FUNCTION_BLOCK FB_System_WDT_500

VAR_INPUT
	Betrieb_Anford_auto				: BOOL;
	Freigabe_Deakt_auto 			: BOOL;
	Regelung_Modus_auto				: USINT;
	Regelung_Nachtabs_auto			: BOOL;
	Regelung_Sollw_auto				: REAL;
	Temp_Rueckl_Wand_Ost_Sektor1	: REAL;
	Temp_Rueckl_Wand_Ost_Sektor2	: REAL;
	Temp_Rueckl_Wand_Ost_Sektor3	: REAL;
	Temp_Rueckl_Wand_West_Sektor1	: REAL;
	Temp_Rueckl_Wand_West_Sektor2	: REAL;
	Temp_Rueckl_Wand_West_Sektor3	: REAL;
	Temp_Rueckl_Decke_Ost_Sektor1	: REAL;
	Temp_Rueckl_Decke_Ost_Sektor2	: REAL;
	Temp_Rueckl_Decke_Ost_Sektor3	: REAL;
	Temp_Rueckl_Decke_West_Sektor1	: REAL;
	Temp_Rueckl_Decke_West_Sektor2	: REAL;
	Temp_Rueckl_Decke_West_Sektor3	: REAL;
	Temp_Rueckl_Aussen_Ost			: REAL;
	Temp_Rueckl_Aussen_West			: REAL;
	Temp_AFA_Aussen					: REAL;

END_VAR
VAR_OUTPUT
	{attribute 'OPC.UA.DA' := '1'}Steuerung				: ST_System_WDT_Steuerung;		
	{attribute 'OPC.UA.DA' := '1'}Stellwert				: ST_System_WDT_Stellwert;		
	{attribute 'OPC.UA.DA' := '1'}Zustand					: ST_System_WDT_Zustand;	
	{attribute 'OPC.UA.DA' := '1'}Parameter				: ST_System_WDT_Parameter;		
END_VAR
VAR
	Pumpe_405				: FB_PU;
	Stellventil_401_402		: FB_SVs;
	Stellventil_403_404		: FB_SVs;
	Stellventil_504_505		: FB_SVs_504_505;
	Pumpe_500				: FB_PU;
	Regelventil_500			: FB_RV;
	Regelventil_561			: FB_RV;
	Regelventil_562			: FB_RV;
	Regelventil_563			: FB_RV;
	Regelventil_571			: FB_RV;
	Regelventil_572			: FB_RV;
	Regelventil_573			: FB_RV;
	Regelventil_541			: FB_RV;
	Regelventil_542			: FB_RV;
	Regelventil_543			: FB_RV;
	Regelventil_551			: FB_RV;
	Regelventil_552			: FB_RV;
	Regelventil_553			: FB_RV;

	Zustandscheck			: FB_System_WDT_Zustandscheck;
	Logik					: FB_System_WDT_Logik;
	Ablaufsteuerung			: FB_System_WDT_Ablaufsteuerung;
	Sollwertscheck			: FB_System_WDT_Sollwertscheck;
	Regelung				: FB_System_WDT_Regelung;
	Stellwertscheck			: FB_System_WDT_Stellwertscheck;




END_VAR
VAR // added by the converter: edge detectors and wires of the graphical bodies
    _w1, _w2, _w4, _w6, _w7, _w8, _w9 : ANY;
    _w3, _w5 : BOOL;
END_VAR

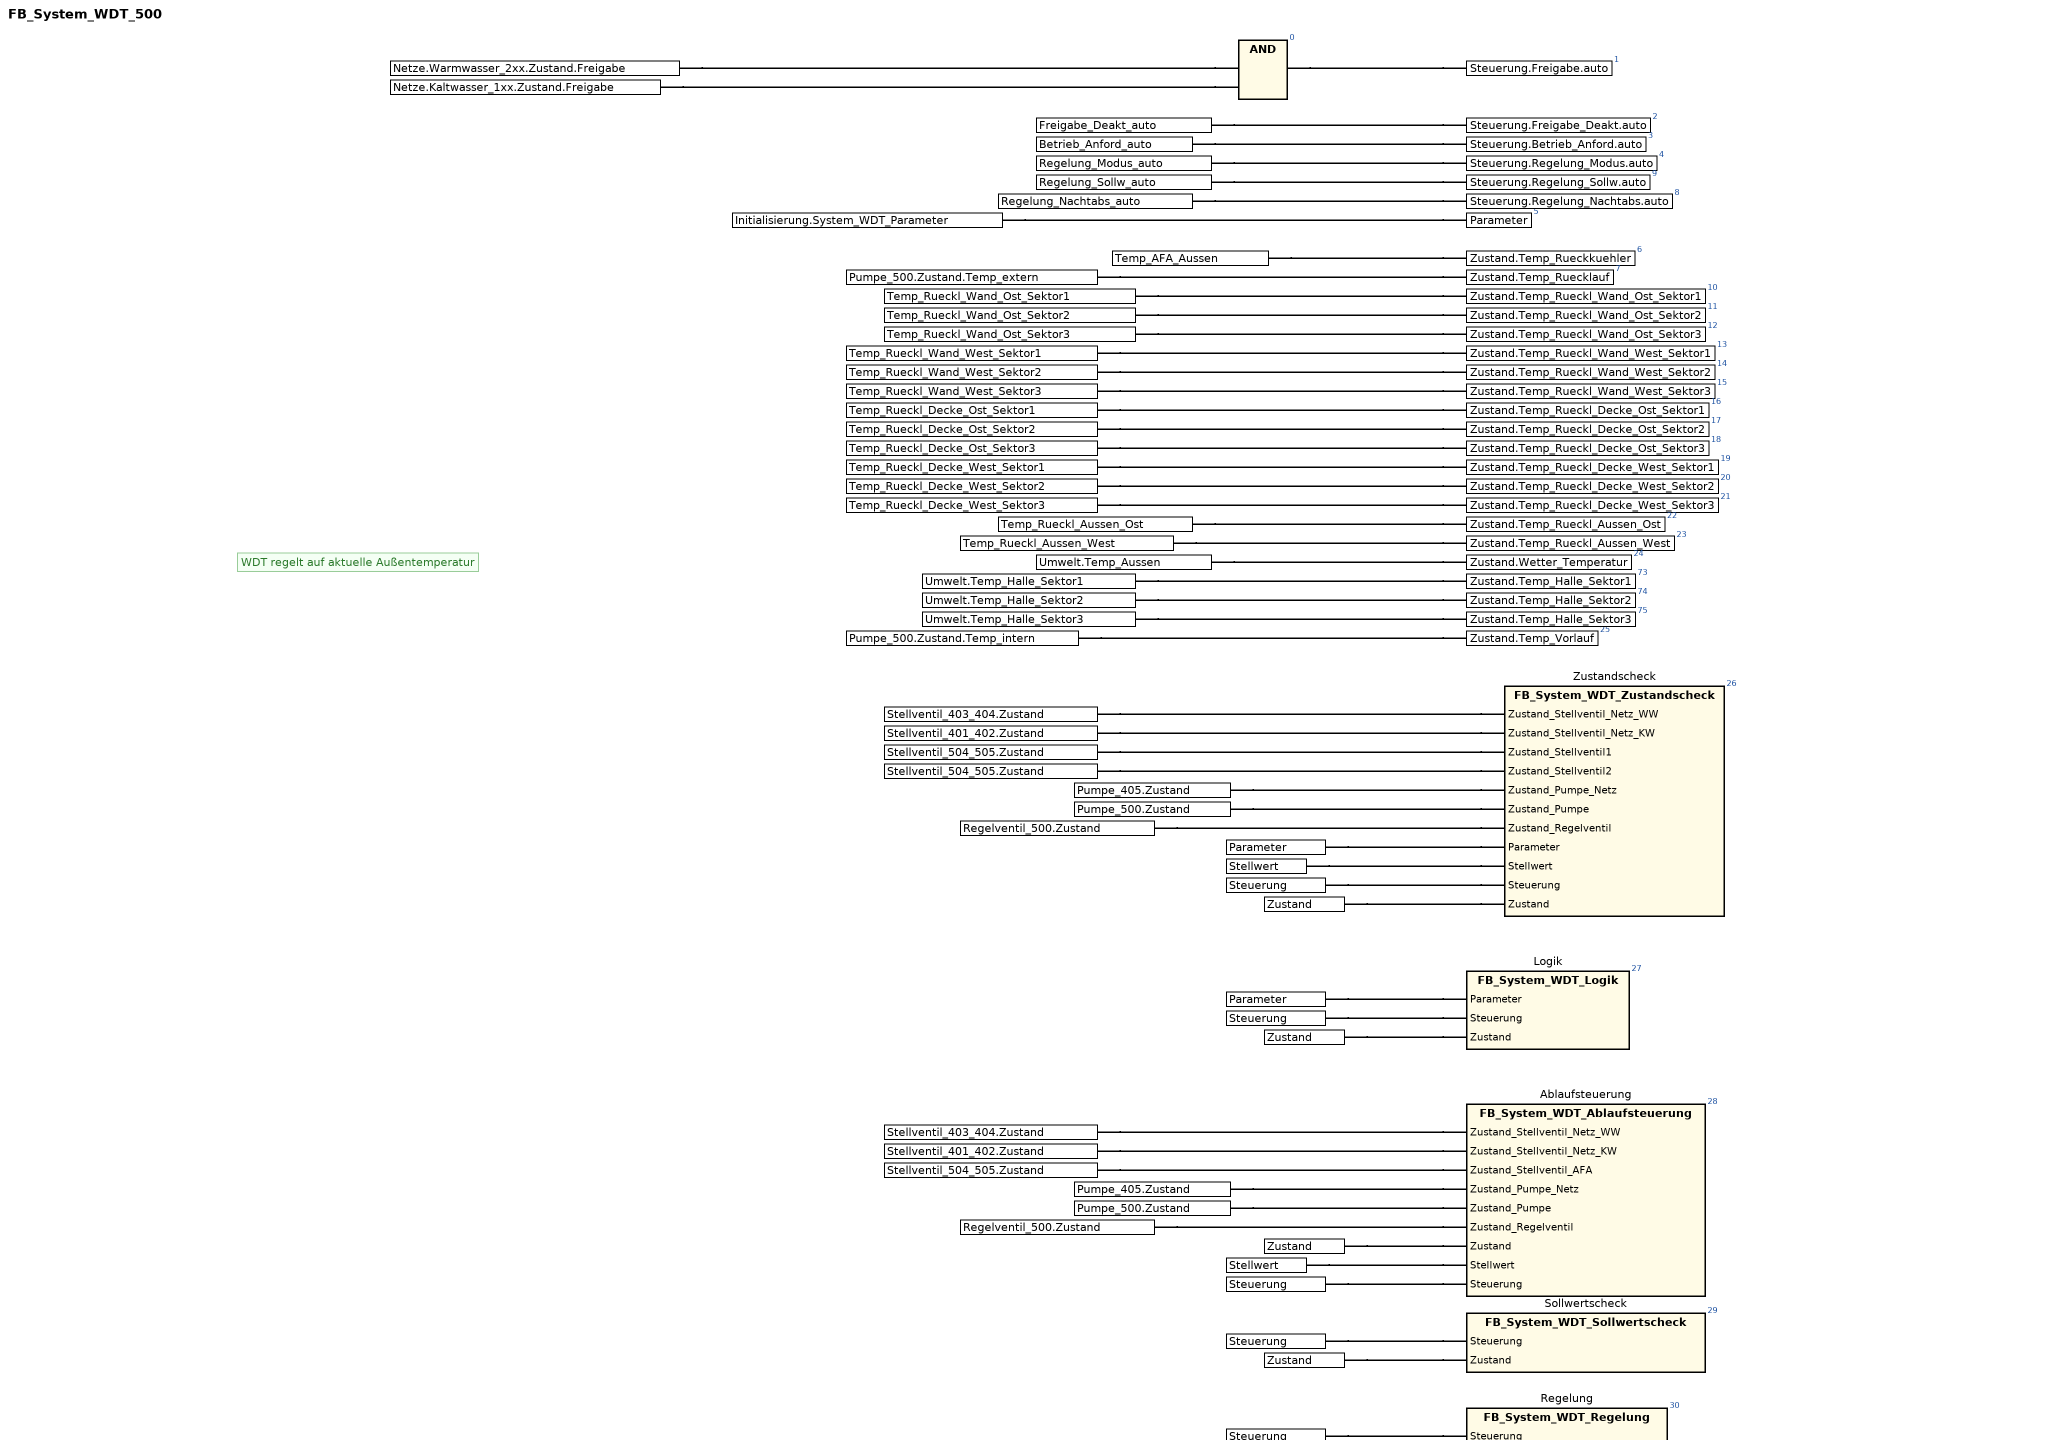
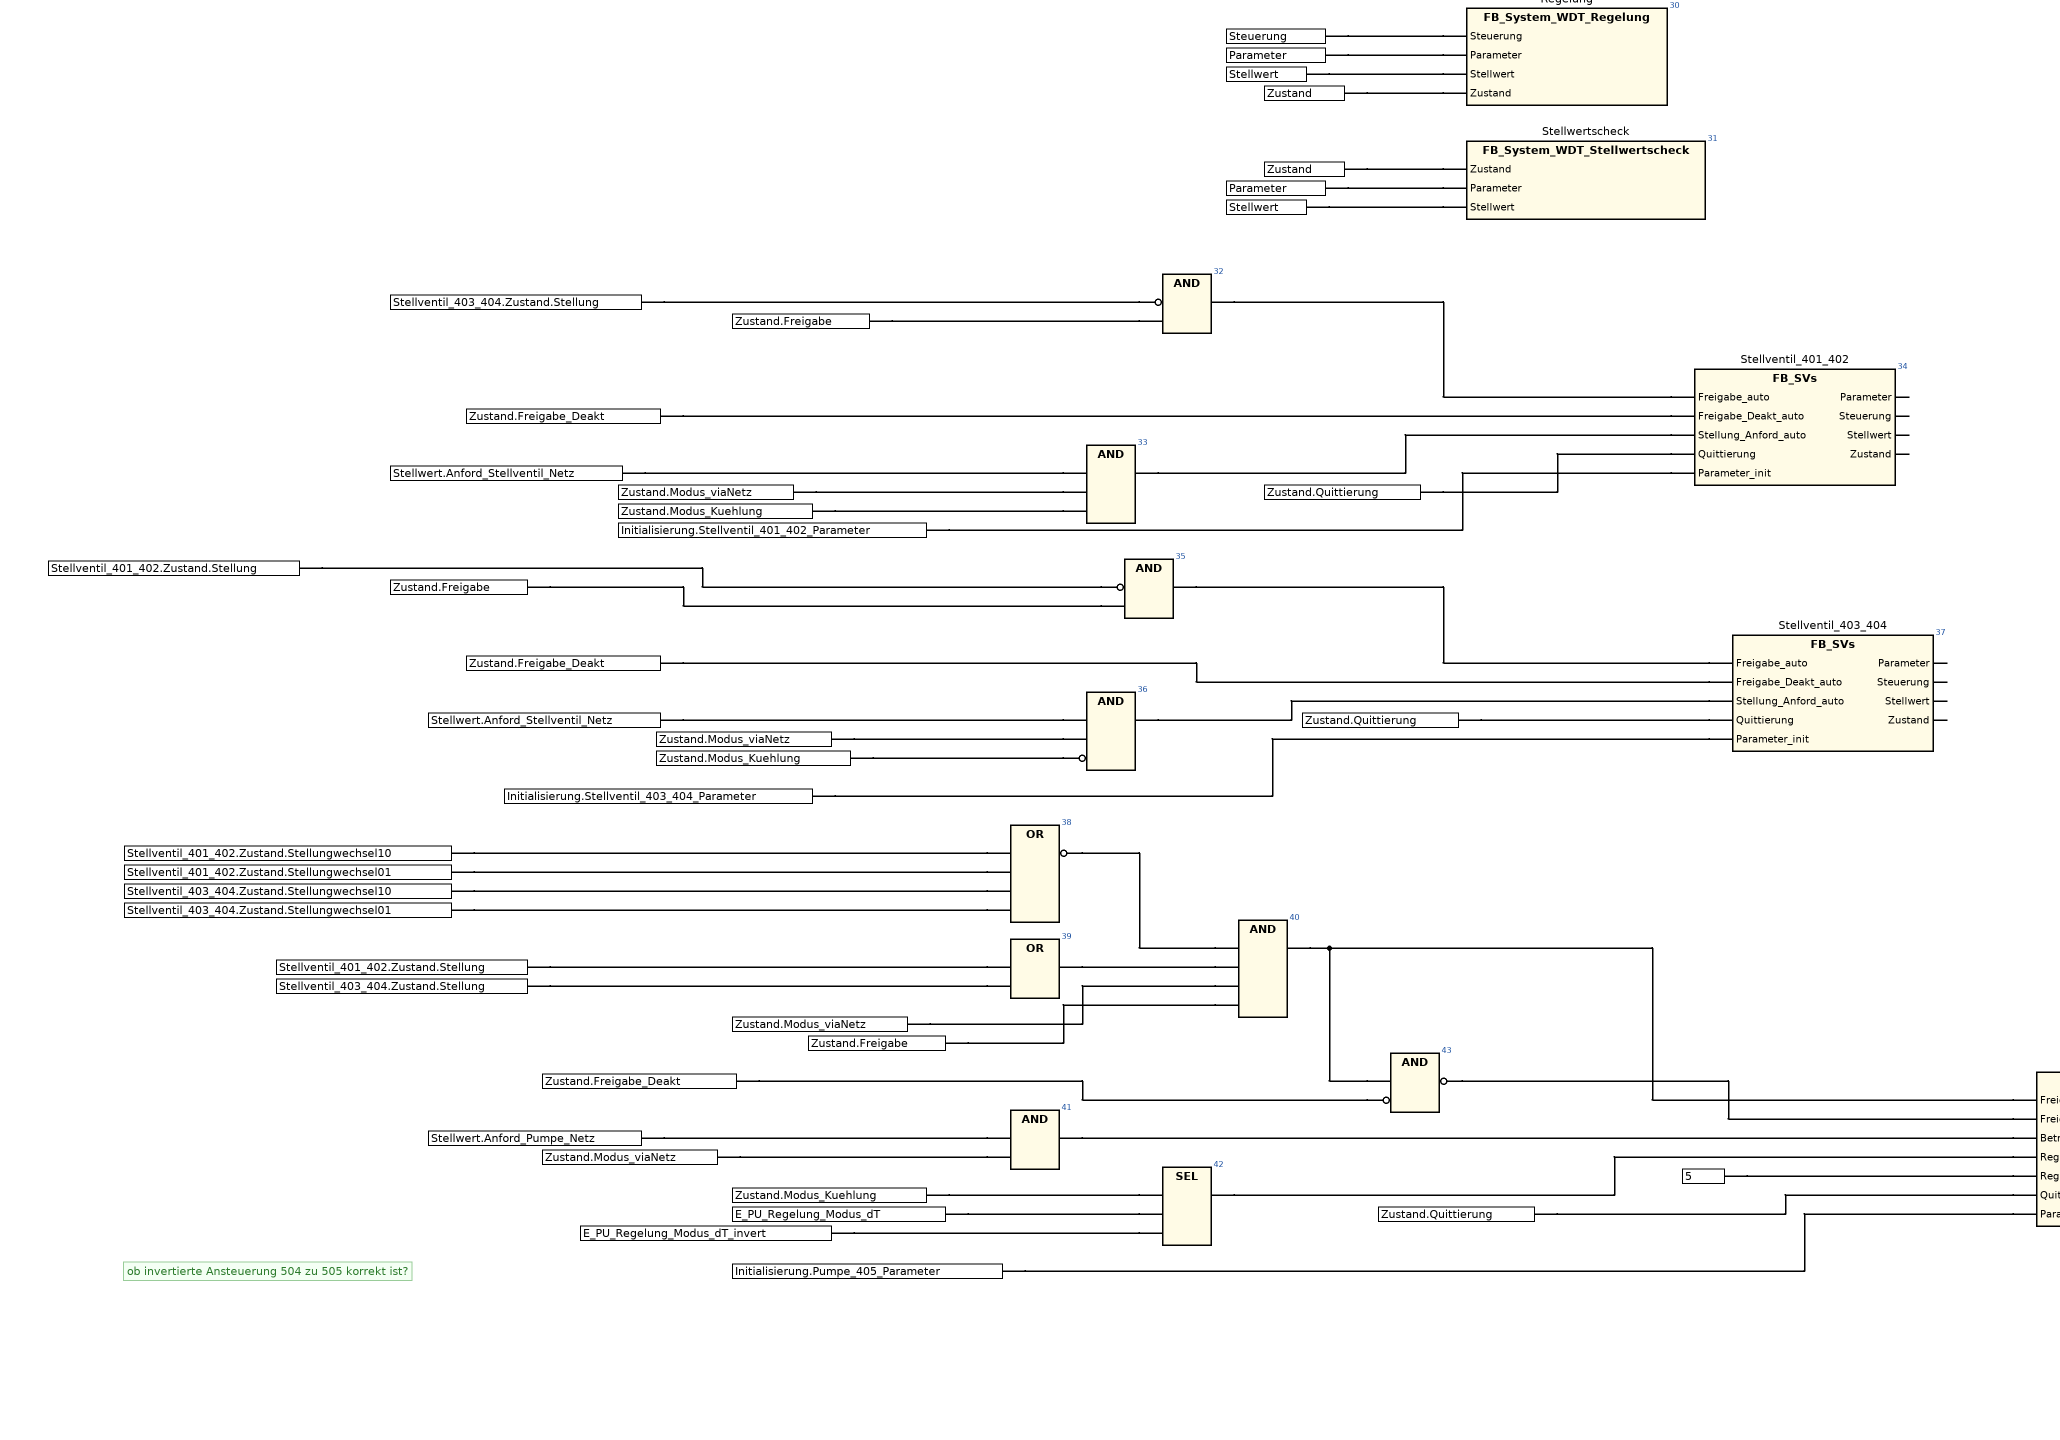
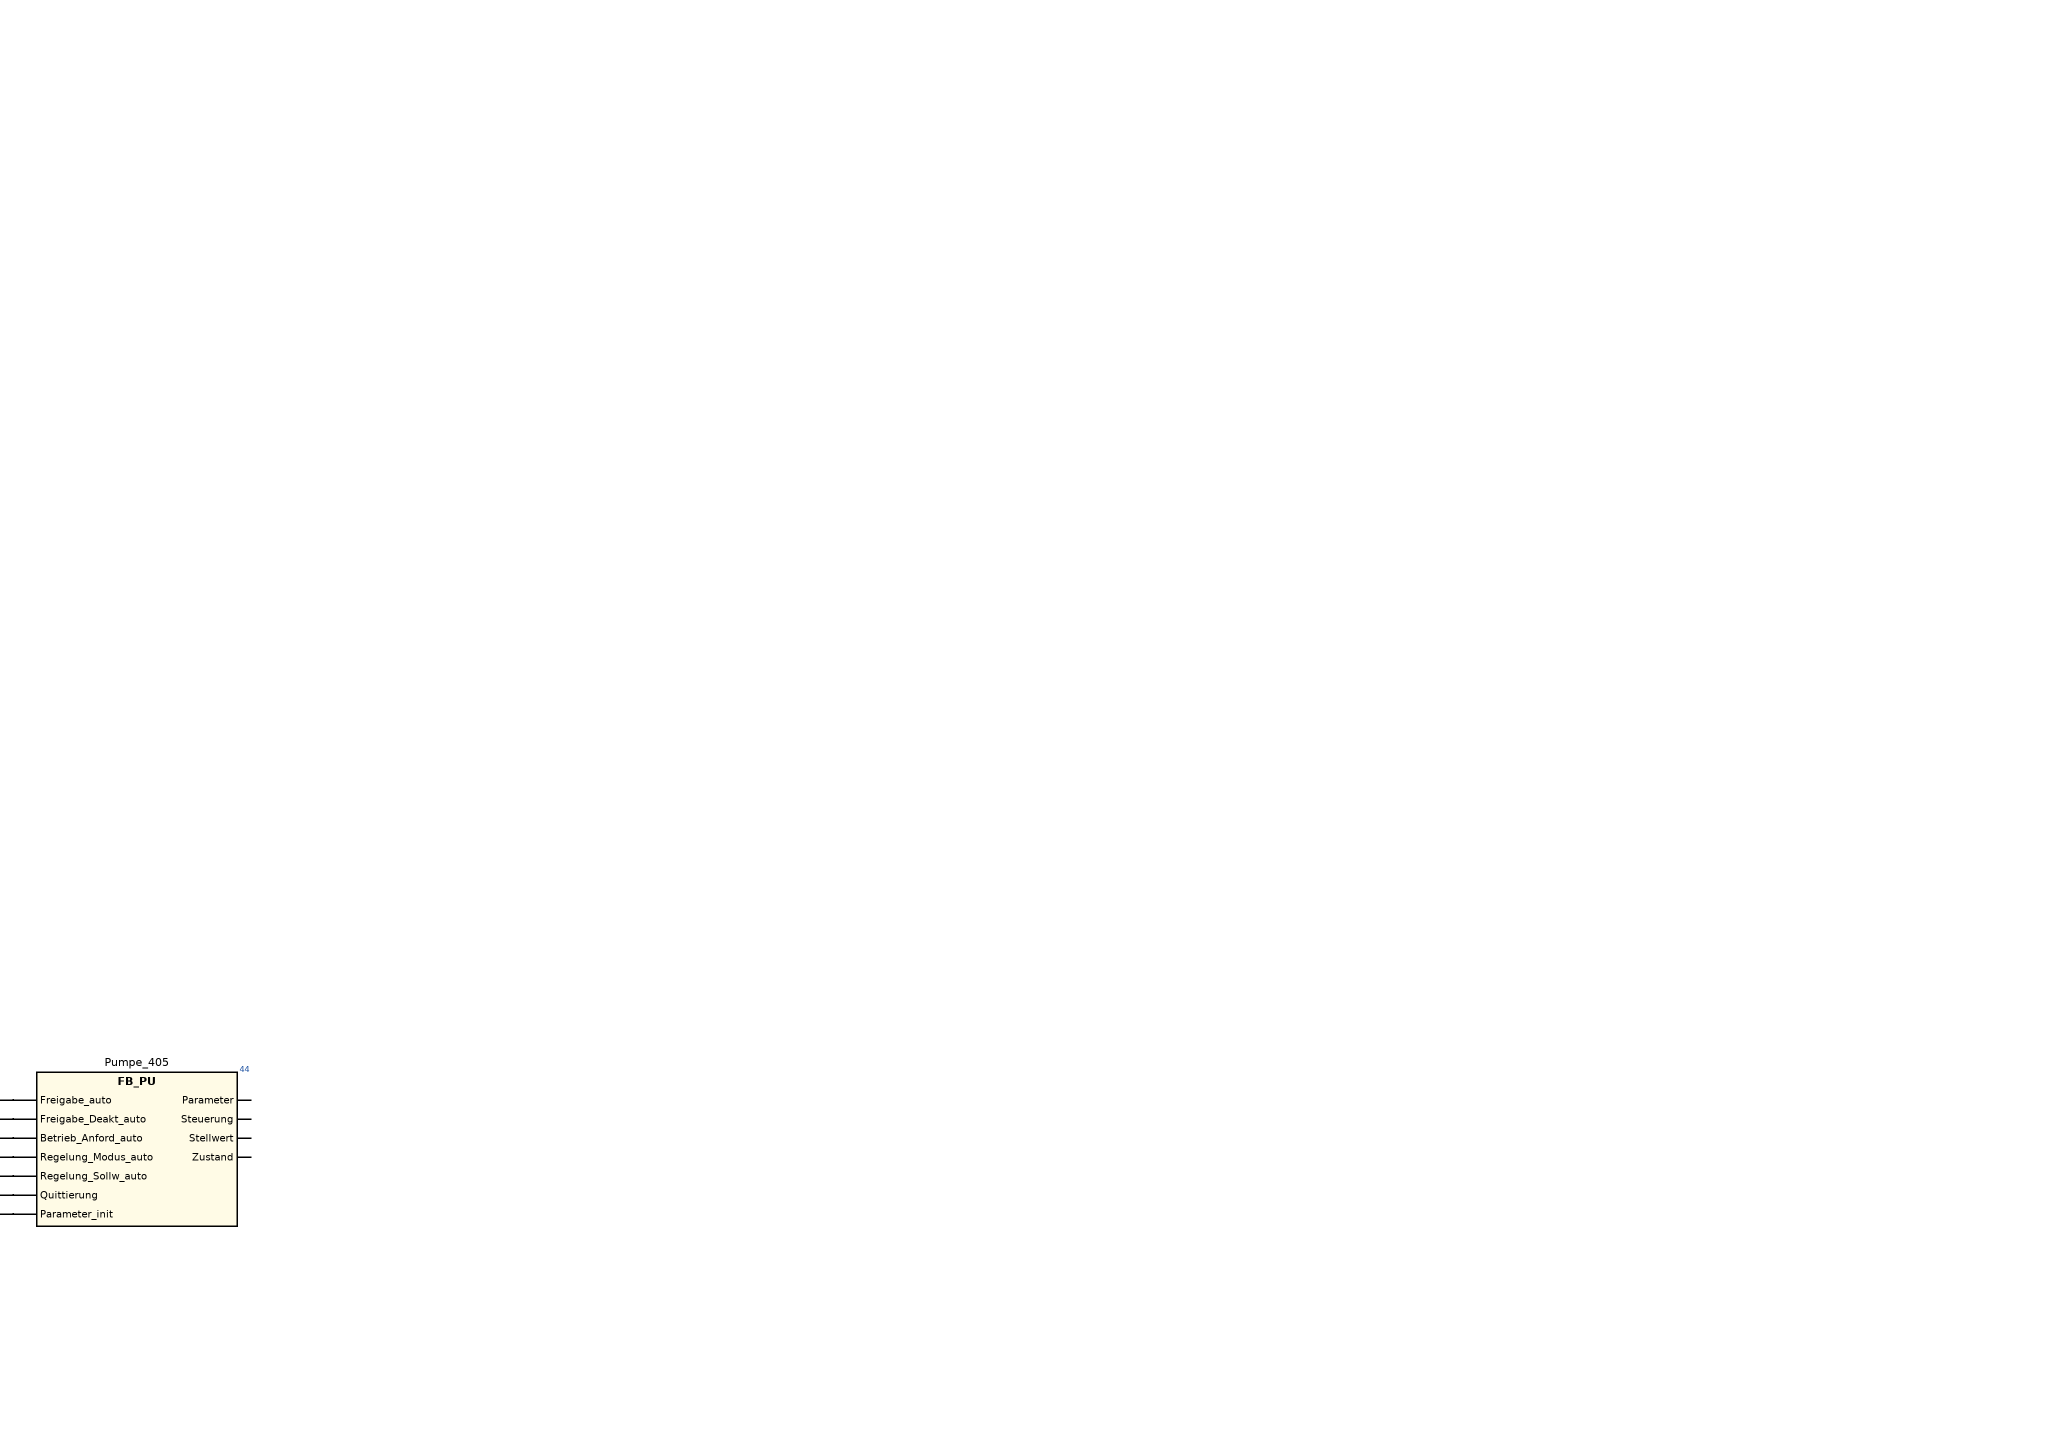
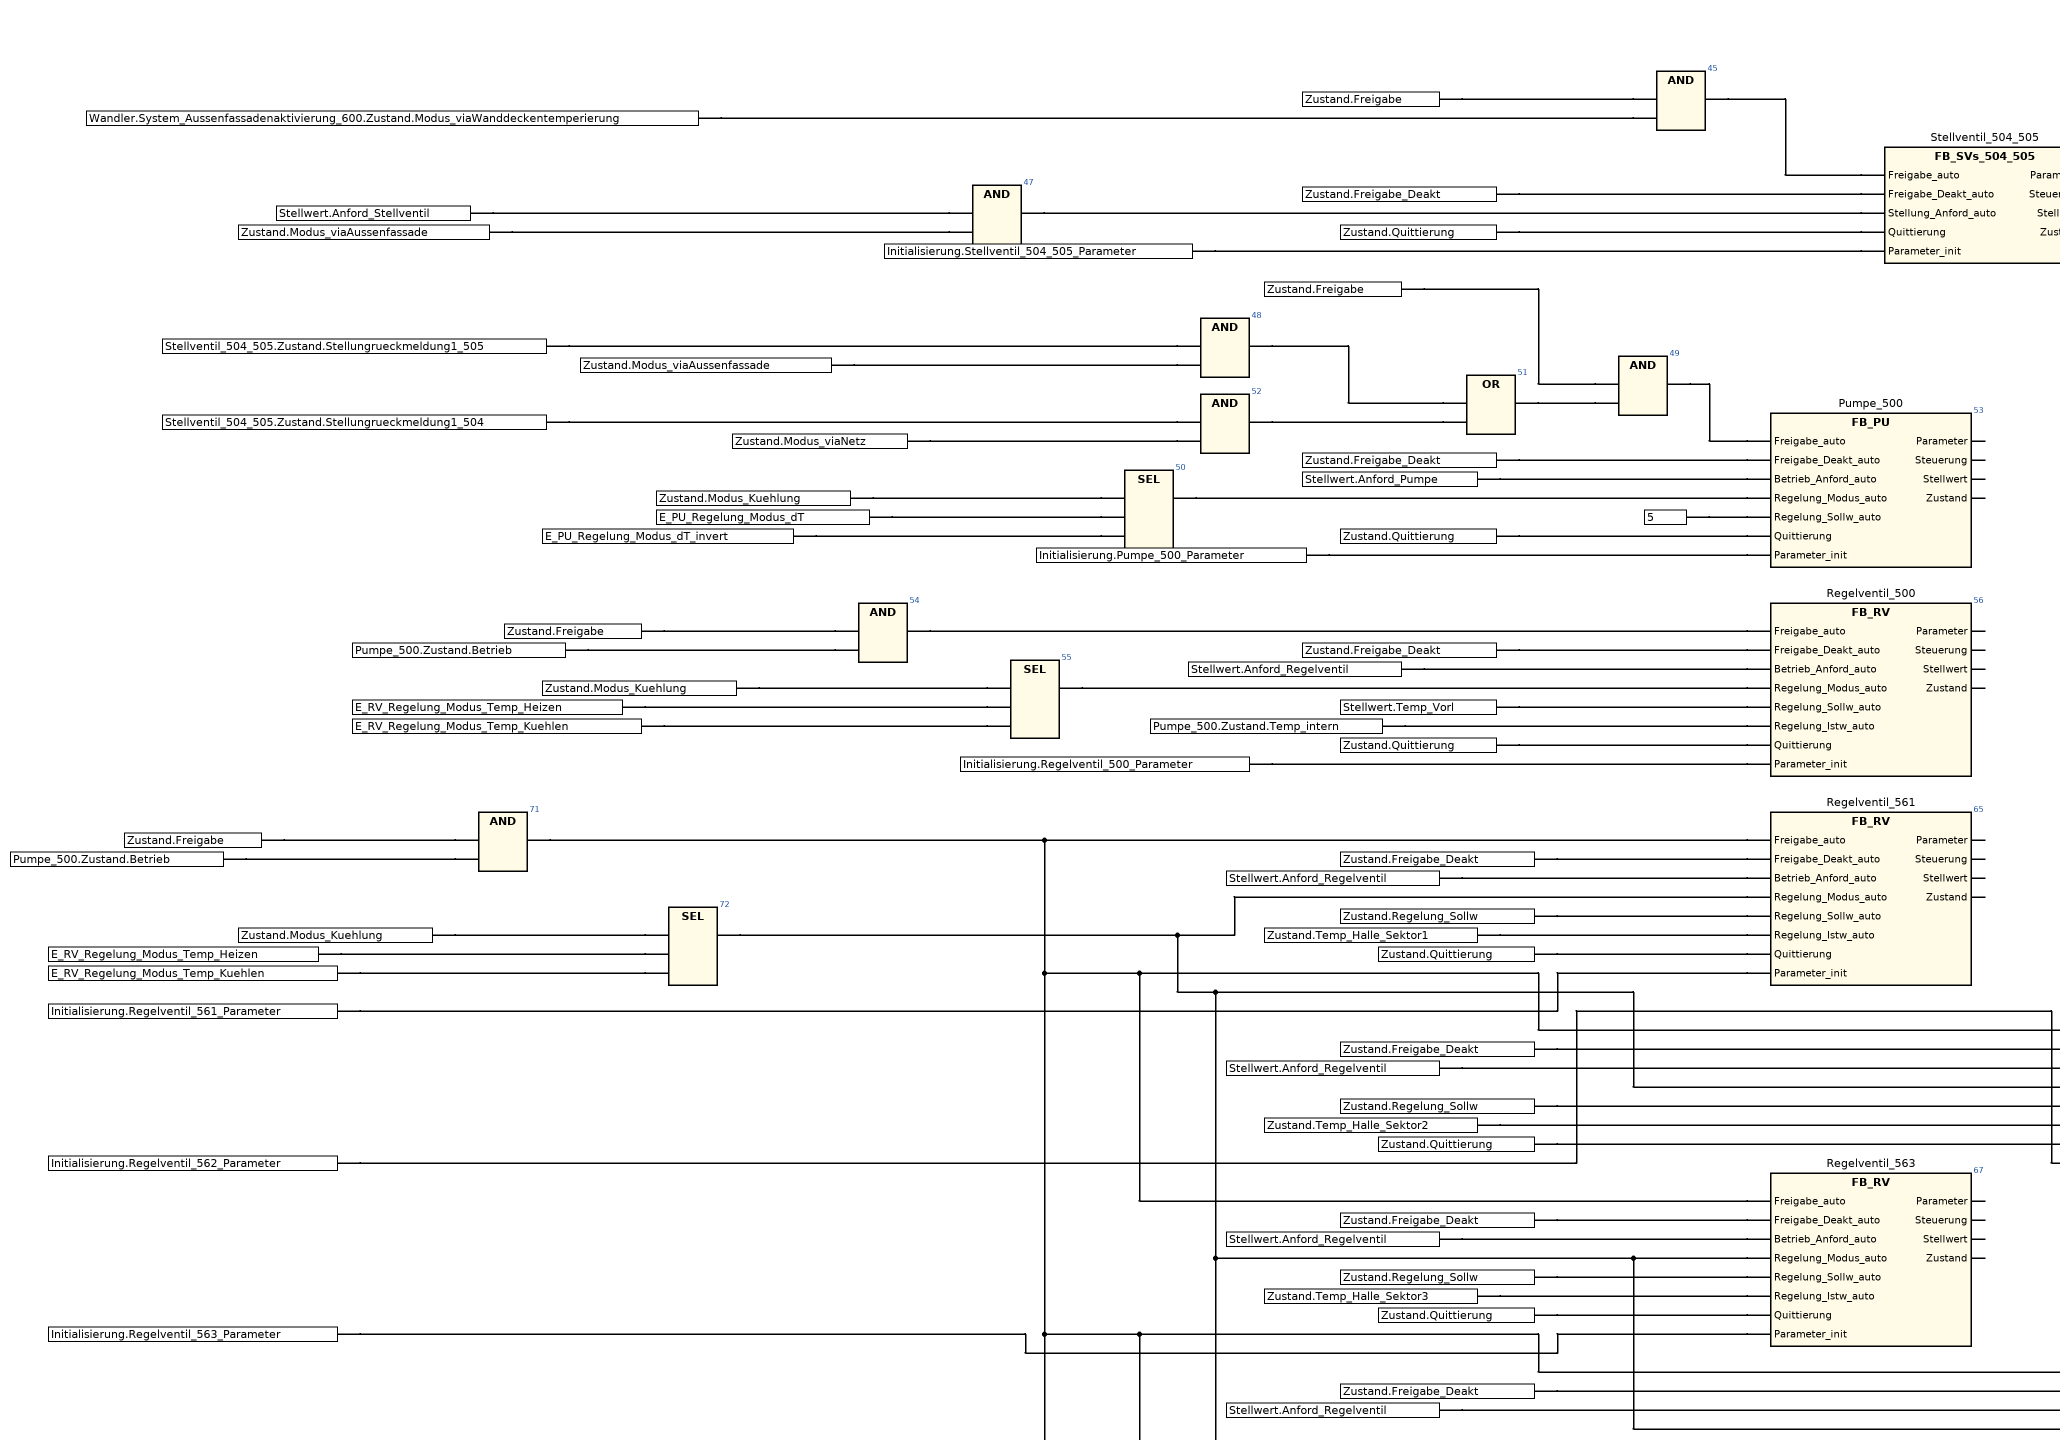
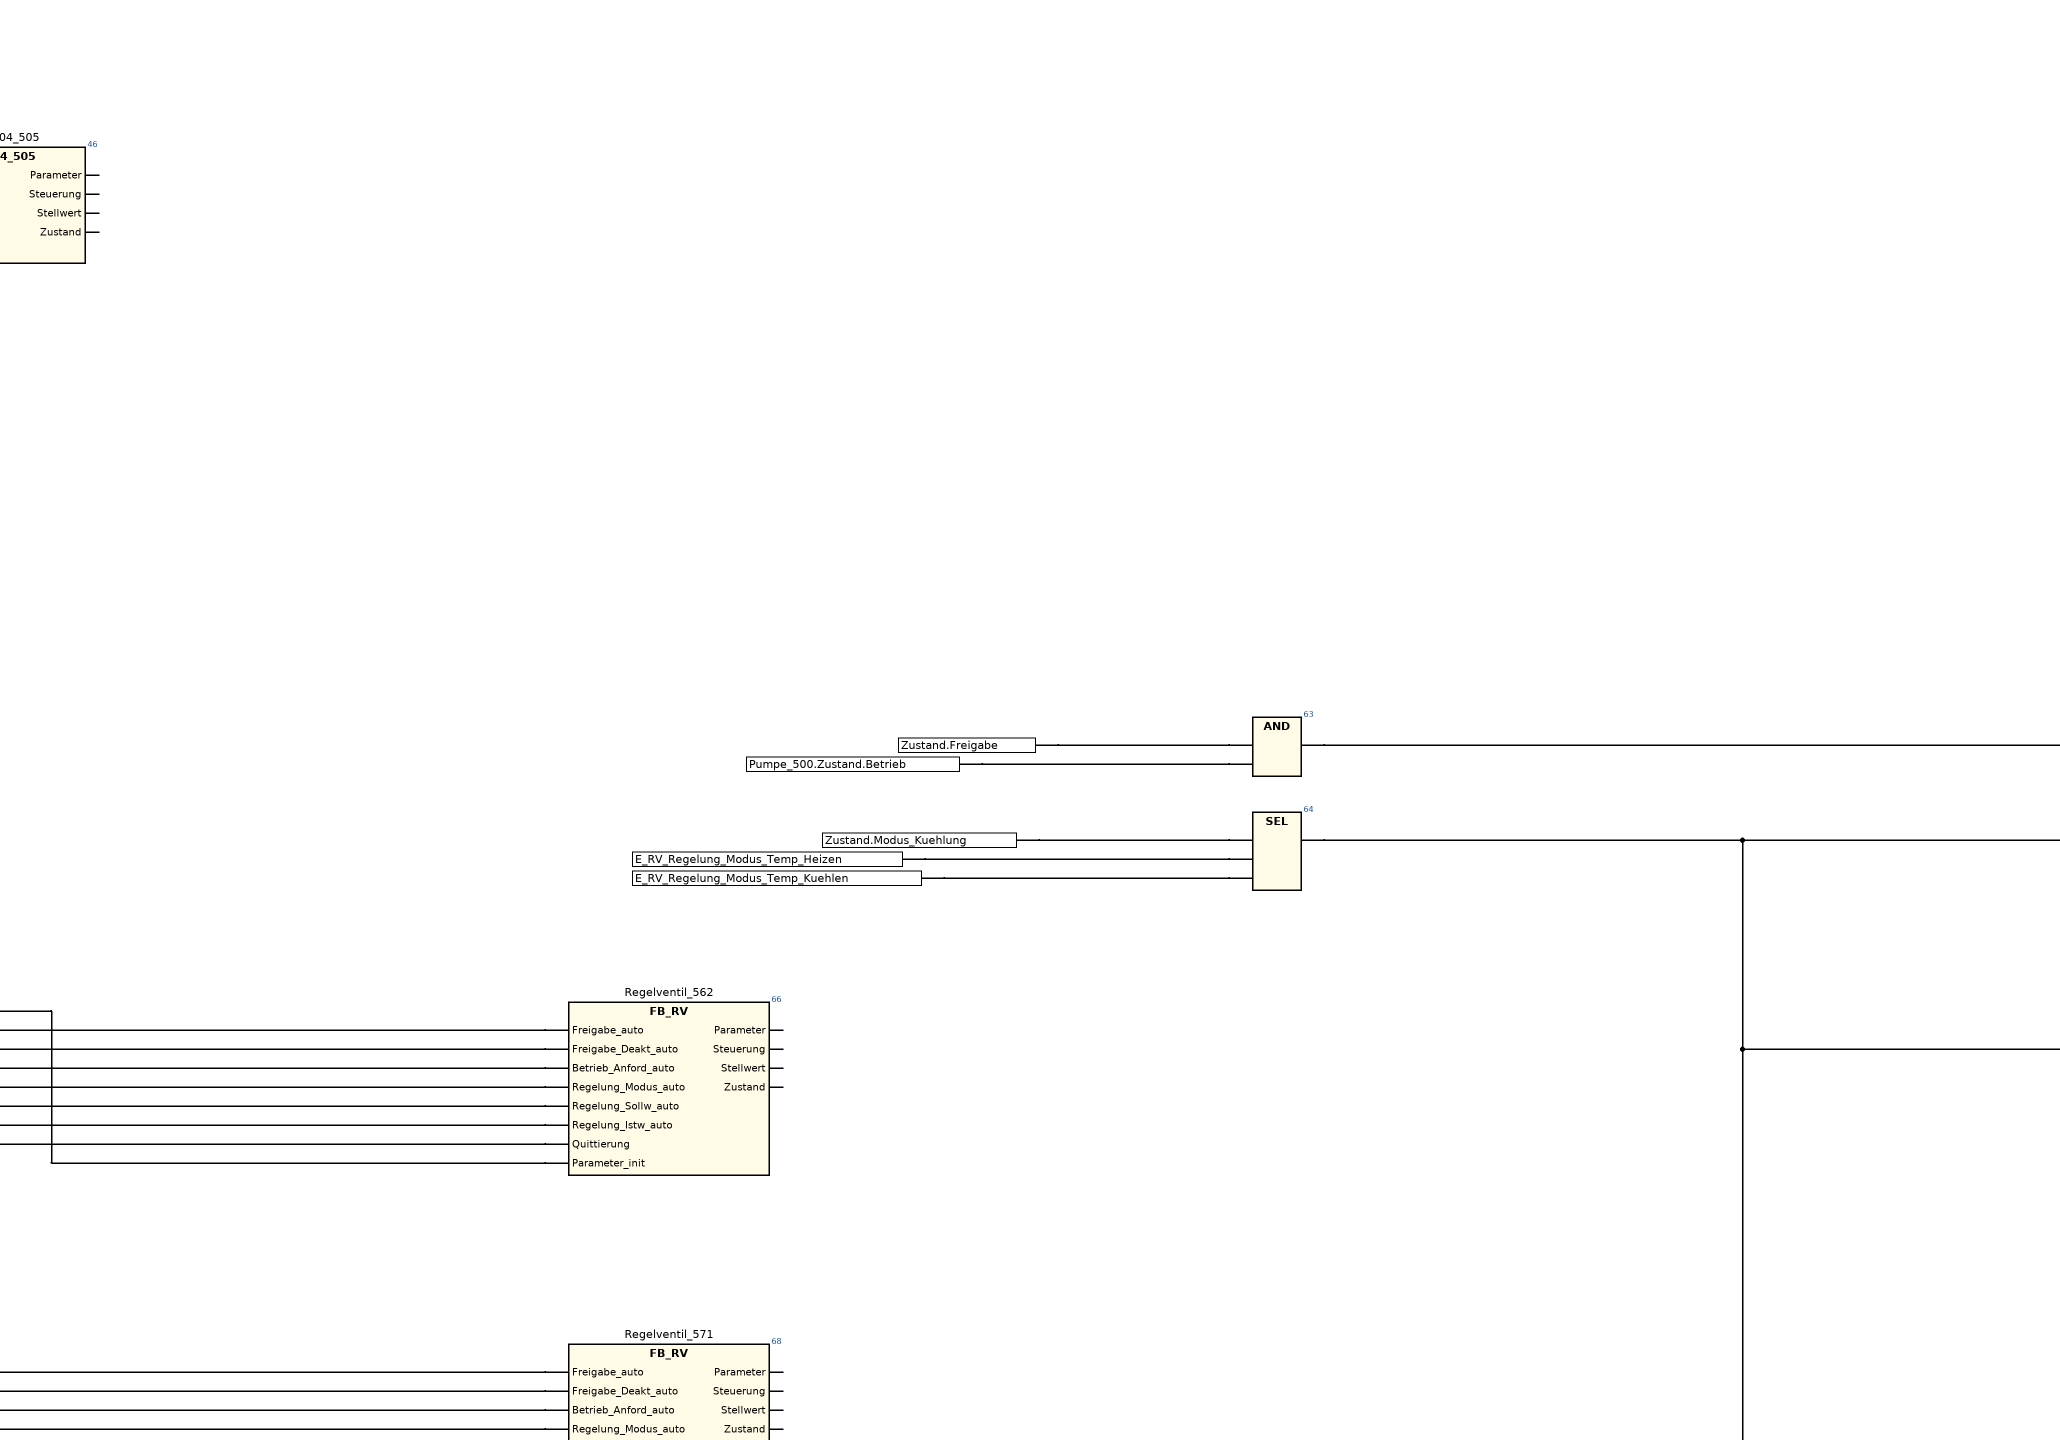
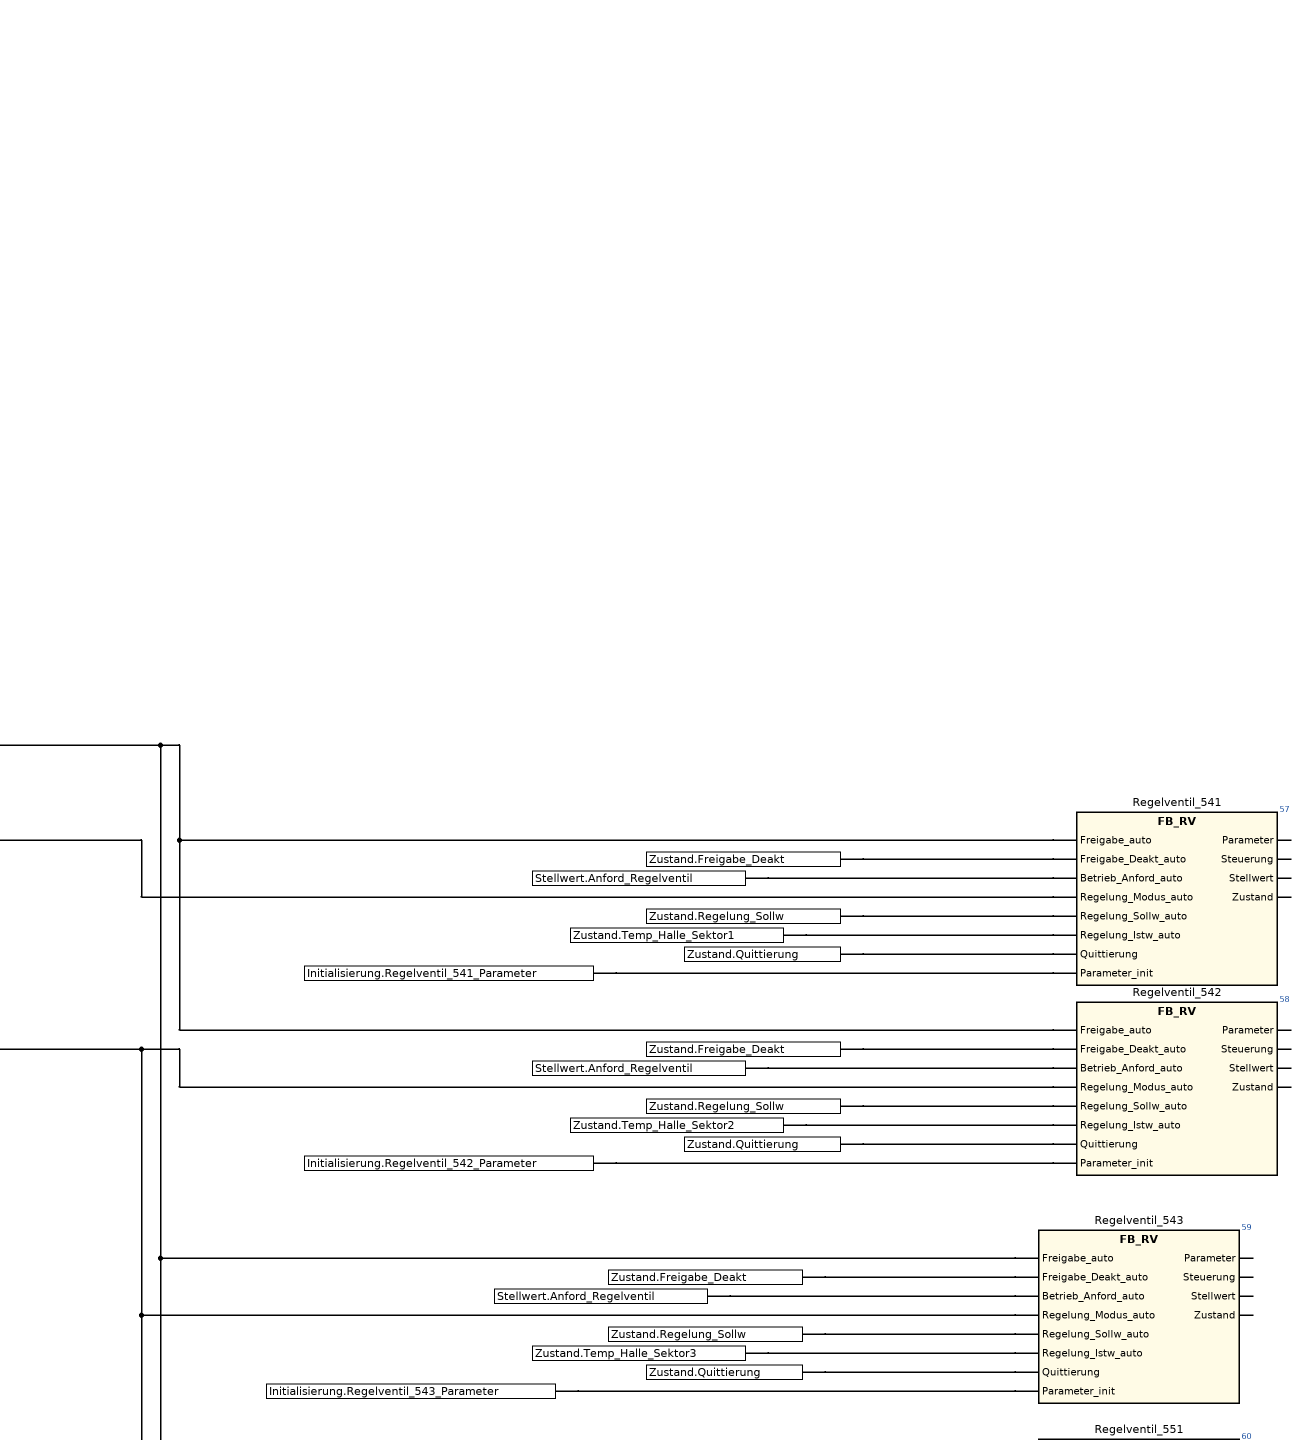
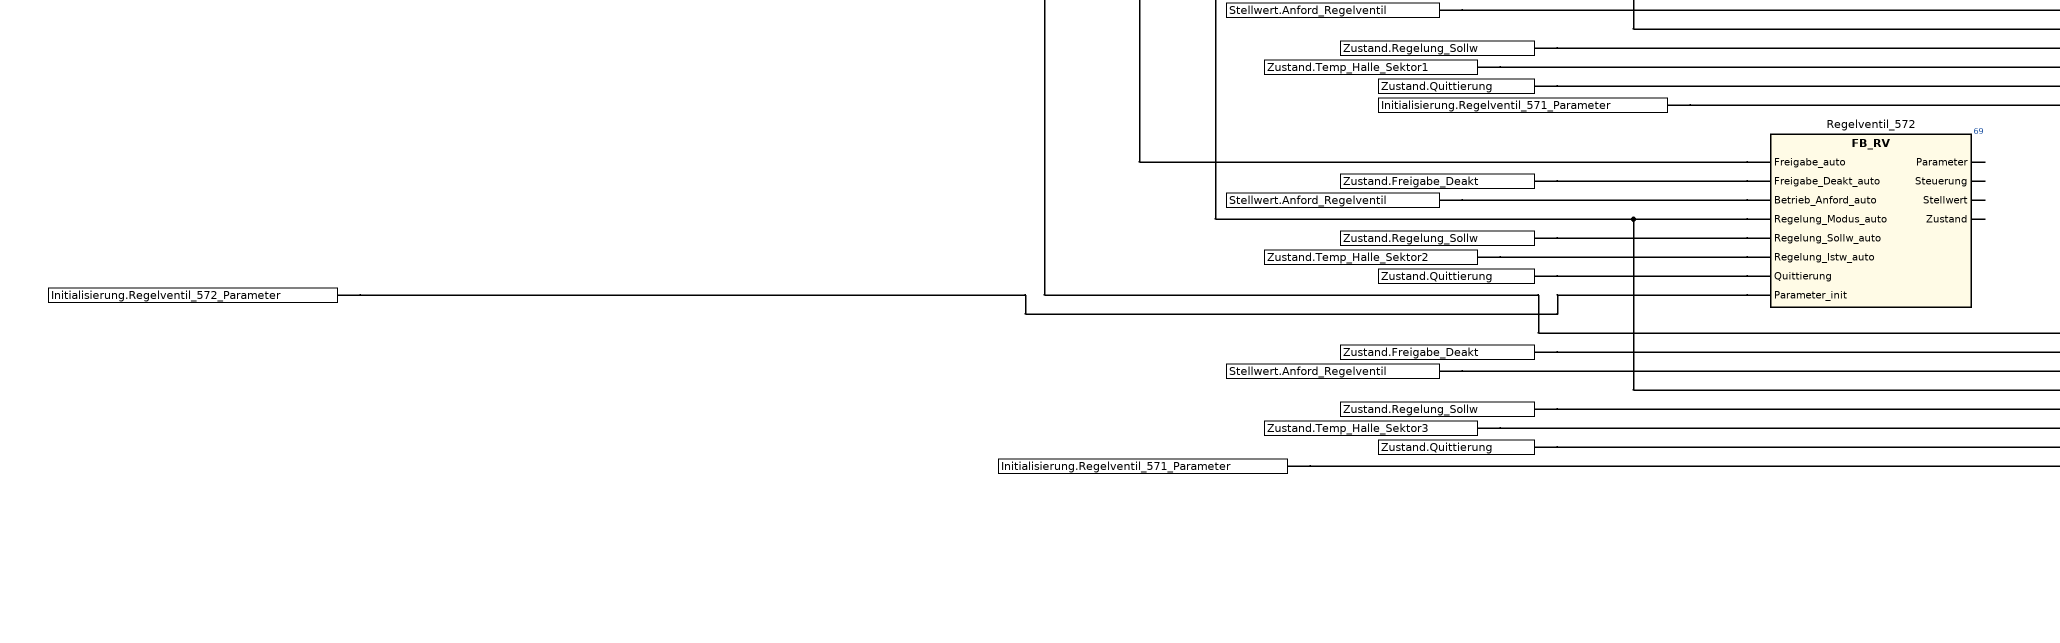
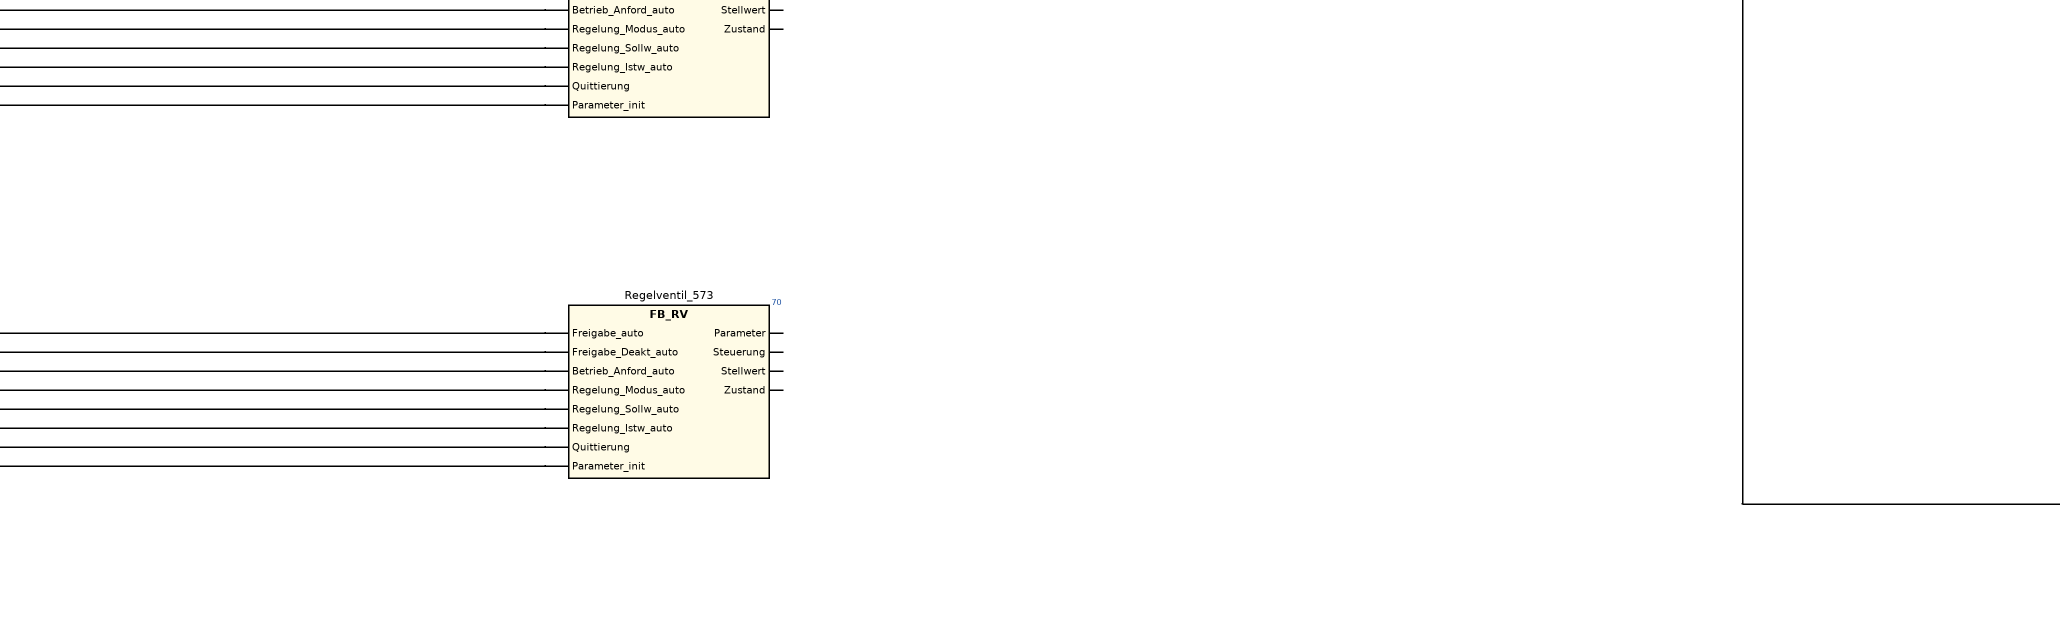
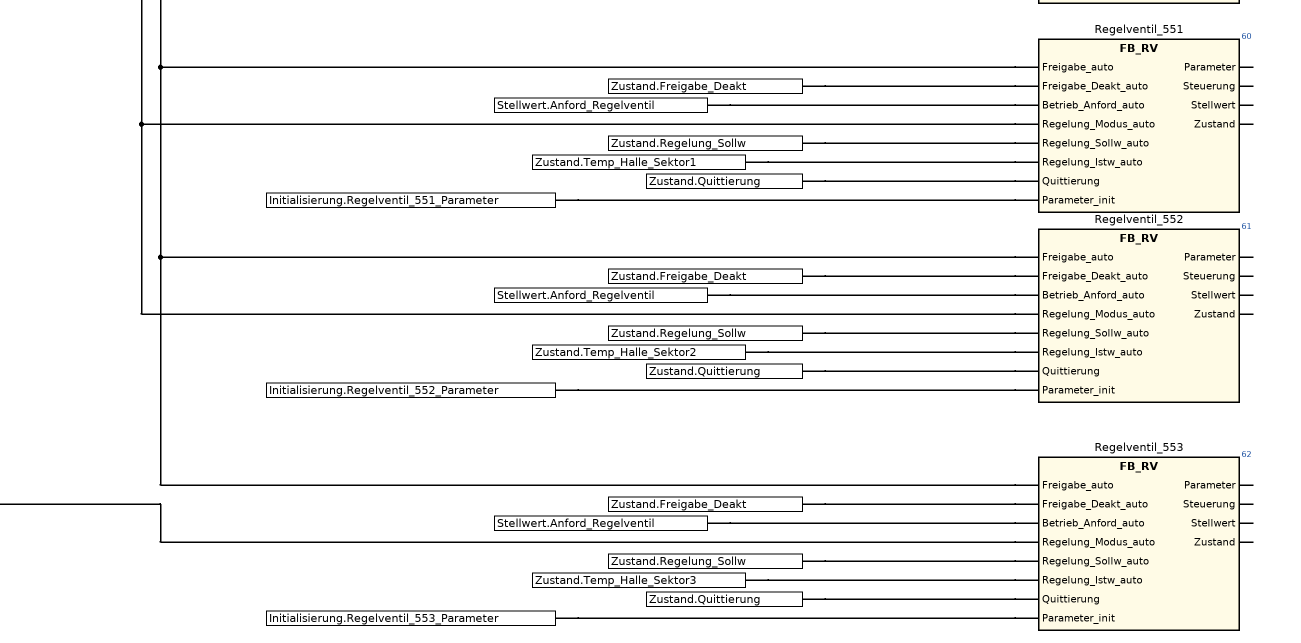
Steuerung.Freigabe.auto := Netze.Warmwasser_2xx.Zustand.Freigabe AND Netze.Kaltwasser_1xx.Zustand.Freigabe;
Steuerung.Freigabe_Deakt.auto := Freigabe_Deakt_auto;
Steuerung.Betrieb_Anford.auto := Betrieb_Anford_auto;
Steuerung.Regelung_Modus.auto := Regelung_Modus_auto;
Parameter := Initialisierung.System_WDT_Parameter;
Zustand.Temp_Rueckkuehler := Temp_AFA_Aussen;
Zustand.Temp_Ruecklauf := Pumpe_500.Zustand.Temp_extern;
Steuerung.Regelung_Nachtabs.auto := Regelung_Nachtabs_auto;
Steuerung.Regelung_Sollw.auto := Regelung_Sollw_auto;
Zustand.Temp_Rueckl_Wand_Ost_Sektor1 := Temp_Rueckl_Wand_Ost_Sektor1;
Zustand.Temp_Rueckl_Wand_Ost_Sektor2 := Temp_Rueckl_Wand_Ost_Sektor2;
Zustand.Temp_Rueckl_Wand_Ost_Sektor3 := Temp_Rueckl_Wand_Ost_Sektor3;
Zustand.Temp_Rueckl_Wand_West_Sektor1 := Temp_Rueckl_Wand_West_Sektor1;
Zustand.Temp_Rueckl_Wand_West_Sektor2 := Temp_Rueckl_Wand_West_Sektor2;
Zustand.Temp_Rueckl_Wand_West_Sektor3 := Temp_Rueckl_Wand_West_Sektor3;
Zustand.Temp_Rueckl_Decke_Ost_Sektor1 := Temp_Rueckl_Decke_Ost_Sektor1;
Zustand.Temp_Rueckl_Decke_Ost_Sektor2 := Temp_Rueckl_Decke_Ost_Sektor2;
Zustand.Temp_Rueckl_Decke_Ost_Sektor3 := Temp_Rueckl_Decke_Ost_Sektor3;
Zustand.Temp_Rueckl_Decke_West_Sektor1 := Temp_Rueckl_Decke_West_Sektor1;
Zustand.Temp_Rueckl_Decke_West_Sektor2 := Temp_Rueckl_Decke_West_Sektor2;
Zustand.Temp_Rueckl_Decke_West_Sektor3 := Temp_Rueckl_Decke_West_Sektor3;
Zustand.Temp_Rueckl_Aussen_Ost := Temp_Rueckl_Aussen_Ost;
Zustand.Temp_Rueckl_Aussen_West := Temp_Rueckl_Aussen_West;
// WDT regelt auf aktuelle Außentemperatur
Zustand.Wetter_Temperatur := Umwelt.Temp_Aussen;
Zustand.Temp_Vorlauf := Pumpe_500.Zustand.Temp_intern;
Zustandscheck(
    Zustand_Stellventil_Netz_WW := Stellventil_403_404.Zustand,
    Zustand_Stellventil_Netz_KW := Stellventil_401_402.Zustand,
    Zustand_Stellventil1 := Stellventil_504_505.Zustand,
    Zustand_Stellventil2 := Stellventil_504_505.Zustand,
    Zustand_Pumpe_Netz := Pumpe_405.Zustand,
    Zustand_Pumpe := Pumpe_500.Zustand,
    Zustand_Regelventil := Regelventil_500.Zustand,
    Parameter := Parameter,
    Stellwert := Stellwert,
    Steuerung := Steuerung,
    Zustand := Zustand); // FB_System_WDT_Zustandscheck
Logik(Parameter := Parameter, Steuerung := Steuerung, Zustand := Zustand); // FB_System_WDT_Logik
Ablaufsteuerung(
    Zustand_Stellventil_Netz_WW := Stellventil_403_404.Zustand,
    Zustand_Stellventil_Netz_KW := Stellventil_401_402.Zustand,
    Zustand_Stellventil_AFA := Stellventil_504_505.Zustand,
    Zustand_Pumpe_Netz := Pumpe_405.Zustand,
    Zustand_Pumpe := Pumpe_500.Zustand,
    Zustand_Regelventil := Regelventil_500.Zustand,
    Zustand := Zustand,
    Stellwert := Stellwert,
    Steuerung := Steuerung); // FB_System_WDT_Ablaufsteuerung
Sollwertscheck(Steuerung := Steuerung, Zustand := Zustand); // FB_System_WDT_Sollwertscheck
Regelung(Steuerung := Steuerung, Parameter := Parameter, Stellwert := Stellwert, Zustand := Zustand); // FB_System_WDT_Regelung
Stellwertscheck(Zustand := Zustand, Parameter := Parameter, Stellwert := Stellwert); // FB_System_WDT_Stellwertscheck
Stellventil_401_402(
    Freigabe_auto := NOT Stellventil_403_404.Zustand.Stellung AND Zustand.Freigabe,
    Freigabe_Deakt_auto := Zustand.Freigabe_Deakt,
    Stellung_Anford_auto := Stellwert.Anford_Stellventil_Netz AND Zustand.Modus_viaNetz AND Zustand.Modus_Kuehlung,
    Quittierung := Zustand.Quittierung,
    Parameter_init := Initialisierung.Stellventil_401_402_Parameter); // FB_SVs
Stellventil_403_404(
    Freigabe_auto := NOT Stellventil_401_402.Zustand.Stellung AND Zustand.Freigabe,
    Freigabe_Deakt_auto := Zustand.Freigabe_Deakt,
    Stellung_Anford_auto := Stellwert.Anford_Stellventil_Netz AND Zustand.Modus_viaNetz AND NOT Zustand.Modus_Kuehlung,
    Quittierung := Zustand.Quittierung,
    Parameter_init := Initialisierung.Stellventil_403_404_Parameter); // FB_SVs
_w1 := NOT (Stellventil_401_402.Zustand.Stellungwechsel10 OR Stellventil_401_402.Zustand.Stellungwechsel01 OR Stellventil_403_404.Zustand.Stellungwechsel10 OR Stellventil_403_404.Zustand.Stellungwechsel01) AND (Stellventil_401_402.Zustand.Stellung OR Stellventil_403_404.Zustand.Stellung) AND Zustand.Modus_viaNetz AND Zustand.Freigabe;
Pumpe_405(
    Freigabe_auto := _w1,
    Freigabe_Deakt_auto := NOT (_w1 AND NOT Zustand.Freigabe_Deakt),
    Betrieb_Anford_auto := Stellwert.Anford_Pumpe_Netz AND Zustand.Modus_viaNetz,
    Regelung_Modus_auto := SEL(Zustand.Modus_Kuehlung, E_PU_Regelung_Modus_dT, E_PU_Regelung_Modus_dT_invert),
    Regelung_Sollw_auto := 5,
    Quittierung := Zustand.Quittierung,
    Parameter_init := Initialisierung.Pumpe_405_Parameter); // FB_PU
Stellventil_504_505(
    Freigabe_auto := Zustand.Freigabe AND Wandler.System_Aussenfassadenaktivierung_600.Zustand.Modus_viaWanddeckentemperierung,
    Freigabe_Deakt_auto := Zustand.Freigabe_Deakt,
    Stellung_Anford_auto := _w2,
    Quittierung := Zustand.Quittierung,
    Parameter_init := Initialisierung.Stellventil_504_505_Parameter); // FB_SVs_504_505
// ob invertierte Ansteuerung 504 zu 505 korrekt ist?
_w2 := Stellwert.Anford_Stellventil AND Zustand.Modus_viaAussenfassade;
_w4 := Zustand.Freigabe AND _w3;
_w3 := Stellventil_504_505.Zustand.Stellungrueckmeldung1_505 AND Zustand.Modus_viaAussenfassade OR _w5;
_w5 := Stellventil_504_505.Zustand.Stellungrueckmeldung1_504 AND Zustand.Modus_viaNetz;
Pumpe_500(
    Freigabe_auto := _w4,
    Freigabe_Deakt_auto := Zustand.Freigabe_Deakt,
    Betrieb_Anford_auto := Stellwert.Anford_Pumpe,
    Regelung_Modus_auto := SEL(Zustand.Modus_Kuehlung, E_PU_Regelung_Modus_dT, E_PU_Regelung_Modus_dT_invert),
    Regelung_Sollw_auto := 5,
    Quittierung := Zustand.Quittierung,
    Parameter_init := Initialisierung.Pumpe_500_Parameter); // FB_PU
Regelventil_500(
    Freigabe_auto := Zustand.Freigabe AND Pumpe_500.Zustand.Betrieb,
    Freigabe_Deakt_auto := Zustand.Freigabe_Deakt,
    Betrieb_Anford_auto := Stellwert.Anford_Regelventil,
    Regelung_Modus_auto := SEL(Zustand.Modus_Kuehlung, E_RV_Regelung_Modus_Temp_Heizen, E_RV_Regelung_Modus_Temp_Kuehlen),
    Regelung_Sollw_auto := Stellwert.Temp_Vorl,
    Regelung_Istw_auto := Pumpe_500.Zustand.Temp_intern,
    Quittierung := Zustand.Quittierung,
    Parameter_init := Initialisierung.Regelventil_500_Parameter); // FB_RV
Regelventil_541(
    Freigabe_auto := _w6,
    Freigabe_Deakt_auto := Zustand.Freigabe_Deakt,
    Betrieb_Anford_auto := Stellwert.Anford_Regelventil,
    Regelung_Modus_auto := _w7,
    Regelung_Sollw_auto := Zustand.Regelung_Sollw,
    Regelung_Istw_auto := Zustand.Temp_Halle_Sektor1,
    Quittierung := Zustand.Quittierung,
    Parameter_init := Initialisierung.Regelventil_541_Parameter); // FB_RV
Regelventil_542(
    Freigabe_auto := _w6,
    Freigabe_Deakt_auto := Zustand.Freigabe_Deakt,
    Betrieb_Anford_auto := Stellwert.Anford_Regelventil,
    Regelung_Modus_auto := _w7,
    Regelung_Sollw_auto := Zustand.Regelung_Sollw,
    Regelung_Istw_auto := Zustand.Temp_Halle_Sektor2,
    Quittierung := Zustand.Quittierung,
    Parameter_init := Initialisierung.Regelventil_542_Parameter); // FB_RV
Regelventil_543(
    Freigabe_auto := _w6,
    Freigabe_Deakt_auto := Zustand.Freigabe_Deakt,
    Betrieb_Anford_auto := Stellwert.Anford_Regelventil,
    Regelung_Modus_auto := _w7,
    Regelung_Sollw_auto := Zustand.Regelung_Sollw,
    Regelung_Istw_auto := Zustand.Temp_Halle_Sektor3,
    Quittierung := Zustand.Quittierung,
    Parameter_init := Initialisierung.Regelventil_543_Parameter); // FB_RV
Regelventil_551(
    Freigabe_auto := _w6,
    Freigabe_Deakt_auto := Zustand.Freigabe_Deakt,
    Betrieb_Anford_auto := Stellwert.Anford_Regelventil,
    Regelung_Modus_auto := _w7,
    Regelung_Sollw_auto := Zustand.Regelung_Sollw,
    Regelung_Istw_auto := Zustand.Temp_Halle_Sektor1,
    Quittierung := Zustand.Quittierung,
    Parameter_init := Initialisierung.Regelventil_551_Parameter); // FB_RV
Regelventil_552(
    Freigabe_auto := _w6,
    Freigabe_Deakt_auto := Zustand.Freigabe_Deakt,
    Betrieb_Anford_auto := Stellwert.Anford_Regelventil,
    Regelung_Modus_auto := _w7,
    Regelung_Sollw_auto := Zustand.Regelung_Sollw,
    Regelung_Istw_auto := Zustand.Temp_Halle_Sektor2,
    Quittierung := Zustand.Quittierung,
    Parameter_init := Initialisierung.Regelventil_552_Parameter); // FB_RV
Regelventil_553(
    Freigabe_auto := _w6,
    Freigabe_Deakt_auto := Zustand.Freigabe_Deakt,
    Betrieb_Anford_auto := Stellwert.Anford_Regelventil,
    Regelung_Modus_auto := _w7,
    Regelung_Sollw_auto := Zustand.Regelung_Sollw,
    Regelung_Istw_auto := Zustand.Temp_Halle_Sektor3,
    Quittierung := Zustand.Quittierung,
    Parameter_init := Initialisierung.Regelventil_553_Parameter); // FB_RV
_w6 := Zustand.Freigabe AND Pumpe_500.Zustand.Betrieb;
_w7 := SEL(Zustand.Modus_Kuehlung, E_RV_Regelung_Modus_Temp_Heizen, E_RV_Regelung_Modus_Temp_Kuehlen);
Regelventil_561(
    Freigabe_auto := _w8,
    Freigabe_Deakt_auto := Zustand.Freigabe_Deakt,
    Betrieb_Anford_auto := Stellwert.Anford_Regelventil,
    Regelung_Modus_auto := _w9,
    Regelung_Sollw_auto := Zustand.Regelung_Sollw,
    Regelung_Istw_auto := Zustand.Temp_Halle_Sektor1,
    Quittierung := Zustand.Quittierung,
    Parameter_init := Initialisierung.Regelventil_561_Parameter); // FB_RV
Regelventil_562(
    Freigabe_auto := _w8,
    Freigabe_Deakt_auto := Zustand.Freigabe_Deakt,
    Betrieb_Anford_auto := Stellwert.Anford_Regelventil,
    Regelung_Modus_auto := _w9,
    Regelung_Sollw_auto := Zustand.Regelung_Sollw,
    Regelung_Istw_auto := Zustand.Temp_Halle_Sektor2,
    Quittierung := Zustand.Quittierung,
    Parameter_init := Initialisierung.Regelventil_562_Parameter); // FB_RV
Regelventil_563(
    Freigabe_auto := _w8,
    Freigabe_Deakt_auto := Zustand.Freigabe_Deakt,
    Betrieb_Anford_auto := Stellwert.Anford_Regelventil,
    Regelung_Modus_auto := _w9,
    Regelung_Sollw_auto := Zustand.Regelung_Sollw,
    Regelung_Istw_auto := Zustand.Temp_Halle_Sektor3,
    Quittierung := Zustand.Quittierung,
    Parameter_init := Initialisierung.Regelventil_563_Parameter); // FB_RV
Regelventil_571(
    Freigabe_auto := _w8,
    Freigabe_Deakt_auto := Zustand.Freigabe_Deakt,
    Betrieb_Anford_auto := Stellwert.Anford_Regelventil,
    Regelung_Modus_auto := _w9,
    Regelung_Sollw_auto := Zustand.Regelung_Sollw,
    Regelung_Istw_auto := Zustand.Temp_Halle_Sektor1,
    Quittierung := Zustand.Quittierung,
    Parameter_init := Initialisierung.Regelventil_571_Parameter); // FB_RV
Regelventil_572(
    Freigabe_auto := _w8,
    Freigabe_Deakt_auto := Zustand.Freigabe_Deakt,
    Betrieb_Anford_auto := Stellwert.Anford_Regelventil,
    Regelung_Modus_auto := _w9,
    Regelung_Sollw_auto := Zustand.Regelung_Sollw,
    Regelung_Istw_auto := Zustand.Temp_Halle_Sektor2,
    Quittierung := Zustand.Quittierung,
    Parameter_init := Initialisierung.Regelventil_572_Parameter); // FB_RV
Regelventil_573(
    Freigabe_auto := _w8,
    Freigabe_Deakt_auto := Zustand.Freigabe_Deakt,
    Betrieb_Anford_auto := Stellwert.Anford_Regelventil,
    Regelung_Modus_auto := _w9,
    Regelung_Sollw_auto := Zustand.Regelung_Sollw,
    Regelung_Istw_auto := Zustand.Temp_Halle_Sektor3,
    Quittierung := Zustand.Quittierung,
    Parameter_init := Initialisierung.Regelventil_571_Parameter); // FB_RV
_w8 := Zustand.Freigabe AND Pumpe_500.Zustand.Betrieb;
_w9 := SEL(Zustand.Modus_Kuehlung, E_RV_Regelung_Modus_Temp_Heizen, E_RV_Regelung_Modus_Temp_Kuehlen);
Zustand.Temp_Halle_Sektor1 := Umwelt.Temp_Halle_Sektor1;
Zustand.Temp_Halle_Sektor2 := Umwelt.Temp_Halle_Sektor2;
Zustand.Temp_Halle_Sektor3 := Umwelt.Temp_Halle_Sektor3;

END_FUNCTION_BLOCK

(* stored: Version 1.1.0.1, ProductVersion 3.1.4024.9
   POU FB_System_WDT_500: Id {d28bc537-bcc8-4f8e-8c91-c50b362e9f5d}, SpecialFunc None *)
